{attribute 'qualified_only'}
{attribute 'strict'}
TYPE GeneralStatus:
( 
	UNKNOWN    := 0,
    READY := 1,
    NOT_READY := 2,
	ERROR := 3
);
END_TYPE

(* stored: Version 1.1.0.1, ProductVersion 3.1.4024.12
   DUT GeneralStatus: Id {b52ea538-2ca0-4b6f-b42f-a96d71adbc3e} *)
